(* PLC project Tc2_Utilities.WORD_TO_FIX16 Demo, tc3-libraries-kb TwinCAT 3.1 *)
(* stored: creationDateTime 2026-05-12T12:00:00, modificationDateTime 2026-05-12T12:00:00 *)

PROGRAM P_Demo_WORD_TO_FIX16
  VAR
    wFromSdo : WORD := 2#0000110010000000;;  (* PDF 示例值 = 12.5 in Q8 *)
    fp8Decoded : T_FIX16;
    lrCheck : LREAL;
    bDecode : BOOL;
  END_VAR

            // ============================================================
// Tc2_Utilities.WORD_TO_FIX16 演示程序（FUNCTION，单周期触发）
// ============================================================
// 场景：EtherCAT SDO 读回 16 位字，重新解读为 Q8 定点。
// 价值：替代 `INT_TO_FIX16(WORD_TO_INT(...), n)` 两层转换。
// 验证步骤：
//   1. 把本 PROGRAM 加到 PlcTask 调用列表
//   2. 编译 + 登录
//   3. 在线把 b... 触发位置 TRUE 一个周期
//   4. 观察输出变量是否符合期望
// ============================================================

IF bDecode THEN
    fp8Decoded := WORD_TO_FIX16(wFromSdo, 8);
    lrCheck    := FIX16_TO_LREAL(fp8Decoded);   // 应为 12.5
    bDecode := FALSE;
END_IF;

          
END_PROGRAM
